KUKA KRL program: Milling_8_4.src

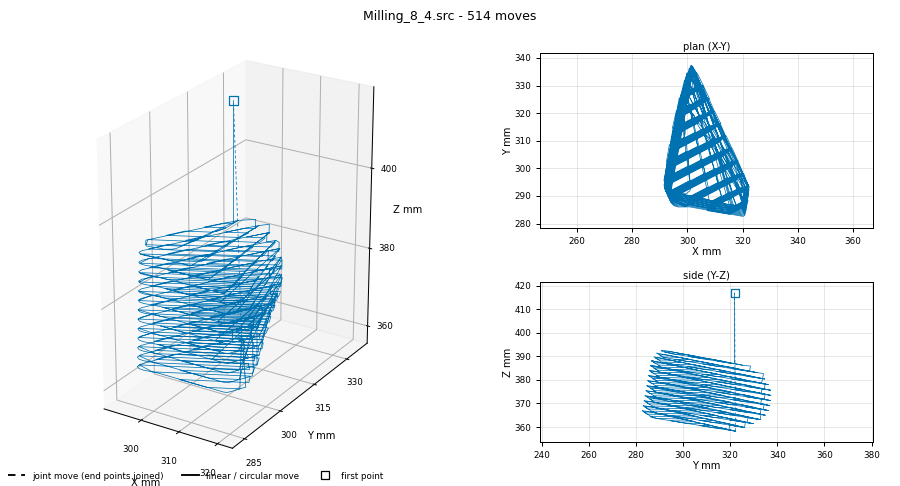
[picture p0: tool path of Milling_8_4.src, 514 of 516 moves have a stored position in this frame; points joined in program order, loops and branches not executed]
&ACCESS RVP
&REL 1
&PARAM TEMPLATE = C:\KRC\Roboter\Template\vorgabe
&PARAM EDITMASK = *
DEF Milling_8_4 ( )


;FOLD INI
;FOLD BASISTECH INI
GLOBAL INTERRUPT DECL 3 WHEN $STOPMESS==TRUE DO IR_STOPM ( )
INTERRUPT ON 3
BAS (#INITMOV,0 )
;ENDFOLD (BASISTECH INI)
;ENDFOLD (INI)

;FOLD STARTPOSITION - BASE IS 0, TOOL IS 5, SPEED IS 15%, POSITION IS A1 5,A2 -90,A3 100,A4 5,A5 -10,A6 -5,E1 0,E2 0,E3 0,E4 0
$BWDSTART = FALSE
PDAT_ACT = {VEL 15,ACC 100,APO_DIST 50}
FDAT_ACT = {TOOL_NO 5,BASE_NO 0,IPO_FRAME #BASE}
BAS (#PTP_PARAMS,15)
PTP  {A1 5,A2 -90,A3 100,A4 5,A5 -10,A6 -5,E1 0,E2 0,E3 0,E4 0}
;ENDFOLD

;FOLD LIN SPEED IS 0.1 m/sec, INTERPOLATION SETTINGS IN FOLD
$VEL.CP=0.1
$ADVANCE=3
;ENDFOLD

BAS(#VEL_PTP,2)
PTP {X 297.852, Y 321.837, Z 416.933, A -65.265, B 78.944, C -140.572, E1 0, E2 0, E3 0, E4 0, S 'B010'}
$VEL.CP=0.012
LIN {X 297.852, Y 321.837, Z 386.933, A -65.265, B 78.944, C -140.572, E1 0, E2 0, E3 0, E4 0}
LIN {X 295.987, Y 320.861, Z 386.954, A -65.265, B 78.944, C -140.572, E1 0, E2 0, E3 0, E4 0}
LIN {X 294.555, Y 314.544, Z 387.958, A -65.265, B 78.944, C -140.572, E1 0, E2 0, E3 0, E4 0}
LIN {X 298.939, Y 316.84, Z 387.909, A -65.265, B 78.944, C -140.572, E1 0, E2 0, E3 0, E4 0}
LIN {X 298.897, Y 311.252, Z 388.897, A -65.265, B 78.944, C -140.572, E1 0, E2 0, E3 0, E4 0}
LIN {X 293.416, Y 308.381, Z 388.959, A -65.265, B 78.944, C -140.572, E1 0, E2 0, E3 0, E4 0}
LIN {X 292.389, Y 302.277, Z 389.958, A -65.265, B 78.944, C -140.572, E1 0, E2 0, E3 0, E4 0}
LIN {X 299.803, Y 306.16, Z 389.875, A -65.265, B 78.944, C -140.572, E1 0, E2 0, E3 0, E4 0}
LIN {X 300.521, Y 300.97, Z 390.855, A -65.265, B 78.944, C -140.572, E1 0, E2 0, E3 0, E4 0}
LIN {X 291.565, Y 296.279, Z 390.955, A -65.265, B 78.944, C -140.572, E1 0, E2 0, E3 0, E4 0}
LIN {X 293.945, Y 291.959, Z 391.916, A -65.265, B 78.944, C -140.572, E1 0, E2 0, E3 0, E4 0}
LIN {X 300.779, Y 295.539, Z 391.84, A -65.265, B 78.944, C -140.572, E1 0, E2 0, E3 0, E4 0}
LIN {X 296.996, Y 325.233, Z 386.261, A -65.265, B 78.944, C -140.572, E1 0, E2 0, E3 0, E4 0}
LIN {X 291.482, Y 295.499, Z 391.087, A -65.265, B 78.944, C -140.572, E1 0, E2 0, E3 0, E4 0}
LIN {X 294.103, Y 291.625, Z 391.989, A -65.265, B 78.944, C -140.572, E1 0, E2 0, E3 0, E4 0}
LIN {X 294.812, Y 290.922, Z 392.171, A -65.265, B 78.944, C -140.572, E1 0, E2 0, E3 0, E4 0}
LIN {X 298.459, Y 290.964, Z 392.462, A -65.265, B 78.944, C -140.572, E1 0, E2 0, E3 0, E4 0}
LIN {X 299.412, Y 290.71, Z 392.585, A -65.265, B 78.944, C -140.572, E1 0, E2 0, E3 0, E4 0}
LIN {X 300.839, Y 291.808, Z 392.507, A -65.265, B 78.944, C -140.572, E1 0, E2 0, E3 0, E4 0}
LIN {X 301.22, Y 292.929, Z 392.339, A -65.265, B 78.944, C -140.572, E1 0, E2 0, E3 0, E4 0}
LIN {X 299.581, Y 309.004, Z 389.352, A -65.265, B 78.944, C -140.572, E1 0, E2 0, E3 0, E4 0}
LIN {X 298.847, Y 311.367, Z 388.873, A -65.265, B 78.944, C -140.572, E1 0, E2 0, E3 0, E4 0}
LIN {X 299.224, Y 312.814, Z 388.647, A -65.265, B 78.944, C -140.572, E1 0, E2 0, E3 0, E4 0}
LIN {X 298.944, Y 316.962, Z 387.888, A -65.265, B 78.944, C -140.572, E1 0, E2 0, E3 0, E4 0}
LIN {X 296.996, Y 325.233, Z 386.261, A -65.265, B 78.944, C -140.572, E1 0, E2 0, E3 0, E4 0}
LIN {X 299.671, Y 328.593, Z 385.883, A -65.265, B 78.944, C -140.572, E1 0, E2 0, E3 0, E4 0}
LIN {X 299.845, Y 328.214, Z 383.749, A -65.265, B 78.944, C -140.572, E1 0, E2 0, E3 0, E4 0}
LIN {X 297.836, Y 327.162, Z 383.772, A -65.265, B 78.944, C -140.572, E1 0, E2 0, E3 0, E4 0}
LIN {X 296.213, Y 320.745, Z 384.778, A -65.265, B 78.944, C -140.572, E1 0, E2 0, E3 0, E4 0}
LIN {X 301.047, Y 323.278, Z 384.724, A -65.265, B 78.944, C -140.572, E1 0, E2 0, E3 0, E4 0}
LIN {X 301.749, Y 318.079, Z 385.704, A -65.265, B 78.944, C -140.572, E1 0, E2 0, E3 0, E4 0}
LIN {X 294.77, Y 314.424, Z 385.782, A -65.265, B 78.944, C -140.572, E1 0, E2 0, E3 0, E4 0}
LIN {X 293.654, Y 308.273, Z 386.783, A -65.265, B 78.944, C -140.572, E1 0, E2 0, E3 0, E4 0}
LIN {X 302.541, Y 312.927, Z 386.683, A -65.265, B 78.944, C -140.572, E1 0, E2 0, E3 0, E4 0}
LIN {X 303.726, Y 307.981, Z 387.658, A -65.265, B 78.944, C -140.572, E1 0, E2 0, E3 0, E4 0}
LIN {X 292.608, Y 302.158, Z 387.782, A -65.265, B 78.944, C -140.572, E1 0, E2 0, E3 0, E4 0}
LIN {X 291.745, Y 296.14, Z 388.78, A -65.265, B 78.944, C -140.572, E1 0, E2 0, E3 0, E4 0}
LIN {X 305.193, Y 303.183, Z 388.629, A -65.265, B 78.944, C -140.572, E1 0, E2 0, E3 0, E4 0}
LIN {X 306.408, Y 298.253, Z 389.603, A -65.265, B 78.944, C -140.572, E1 0, E2 0, E3 0, E4 0}
LIN {X 292.898, Y 291.177, Z 389.755, A -65.265, B 78.944, C -140.572, E1 0, E2 0, E3 0, E4 0}
LIN {X 301.236, Y 289.978, Z 390.649, A -65.265, B 78.944, C -140.572, E1 0, E2 0, E3 0, E4 0}
LIN {X 307.526, Y 293.272, Z 390.579, A -65.265, B 78.944, C -140.572, E1 0, E2 0, E3 0, E4 0}
LIN {X 298.826, Y 331.411, Z 383.099, A -65.265, B 78.944, C -140.572, E1 0, E2 0, E3 0, E4 0}
LIN {X 297.438, Y 325.863, Z 383.97, A -65.265, B 78.944, C -140.572, E1 0, E2 0, E3 0, E4 0}
LIN {X 291.516, Y 293.899, Z 389.159, A -65.265, B 78.944, C -140.572, E1 0, E2 0, E3 0, E4 0}
LIN {X 291.916, Y 292.132, Z 389.505, A -65.265, B 78.944, C -140.572, E1 0, E2 0, E3 0, E4 0}
LIN {X 293.141, Y 290.966, Z 389.812, A -65.265, B 78.944, C -140.572, E1 0, E2 0, E3 0, E4 0}
LIN {X 294.578, Y 290.537, Z 390.005, A -65.265, B 78.944, C -140.572, E1 0, E2 0, E3 0, E4 0}
LIN {X 298.633, Y 290.585, Z 390.328, A -65.265, B 78.944, C -140.572, E1 0, E2 0, E3 0, E4 0}
LIN {X 306.184, Y 288.971, Z 391.232, A -65.265, B 78.944, C -140.572, E1 0, E2 0, E3 0, E4 0}
LIN {X 307.849, Y 288.642, Z 391.427, A -65.265, B 78.944, C -140.572, E1 0, E2 0, E3 0, E4 0}
LIN {X 303.748, Y 307.894, Z 387.675, A -65.265, B 78.944, C -140.572, E1 0, E2 0, E3 0, E4 0}
LIN {X 303.252, Y 309.872, Z 387.283, A -65.265, B 78.944, C -140.572, E1 0, E2 0, E3 0, E4 0}
LIN {X 303.261, Y 309.968, Z 387.267, A -65.265, B 78.944, C -140.572, E1 0, E2 0, E3 0, E4 0}
LIN {X 298.826, Y 331.411, Z 383.099, A -65.265, B 78.944, C -140.572, E1 0, E2 0, E3 0, E4 0}
LIN {X 300.023, Y 334.111, Z 382.718, A -65.265, B 78.944, C -140.572, E1 0, E2 0, E3 0, E4 0}
LIN {X 300.198, Y 333.732, Z 380.584, A -65.265, B 78.944, C -140.572, E1 0, E2 0, E3 0, E4 0}
LIN {X 299.57, Y 333.403, Z 380.591, A -65.265, B 78.944, C -140.572, E1 0, E2 0, E3 0, E4 0}
LIN {X 298.085, Y 327.059, Z 381.596, A -65.265, B 78.944, C -140.572, E1 0, E2 0, E3 0, E4 0}
LIN {X 301.963, Y 329.09, Z 381.552, A -65.265, B 78.944, C -140.572, E1 0, E2 0, E3 0, E4 0}
LIN {X 303.417, Y 324.285, Z 382.524, A -65.265, B 78.944, C -140.572, E1 0, E2 0, E3 0, E4 0}
LIN {X 296.435, Y 320.628, Z 382.602, A -65.265, B 78.944, C -140.572, E1 0, E2 0, E3 0, E4 0}
LIN {X 294.986, Y 314.303, Z 383.606, A -65.265, B 78.944, C -140.572, E1 0, E2 0, E3 0, E4 0}
LIN {X 304.624, Y 319.351, Z 383.498, A -65.265, B 78.944, C -140.572, E1 0, E2 0, E3 0, E4 0}
LIN {X 305.837, Y 314.42, Z 384.473, A -65.265, B 78.944, C -140.572, E1 0, E2 0, E3 0, E4 0}
LIN {X 293.892, Y 308.164, Z 384.606, A -65.265, B 78.944, C -140.572, E1 0, E2 0, E3 0, E4 0}
LIN {X 292.827, Y 302.039, Z 385.606, A -65.265, B 78.944, C -140.572, E1 0, E2 0, E3 0, E4 0}
LIN {X 307.214, Y 309.575, Z 385.445, A -65.265, B 78.944, C -140.572, E1 0, E2 0, E3 0, E4 0}
LIN {X 308.472, Y 304.667, Z 386.419, A -65.265, B 78.944, C -140.572, E1 0, E2 0, E3 0, E4 0}
LIN {X 291.926, Y 296.001, Z 386.604, A -65.265, B 78.944, C -140.572, E1 0, E2 0, E3 0, E4 0}
LIN {X 292.915, Y 290.953, Z 387.581, A -65.265, B 78.944, C -140.572, E1 0, E2 0, E3 0, E4 0}
LIN {X 310.061, Y 299.933, Z 387.389, A -65.265, B 78.944, C -140.572, E1 0, E2 0, E3 0, E4 0}
LIN {X 311.293, Y 295.012, Z 388.363, A -65.265, B 78.944, C -140.572, E1 0, E2 0, E3 0, E4 0}
LIN {X 301.09, Y 289.668, Z 388.477, A -65.265, B 78.944, C -140.572, E1 0, E2 0, E3 0, E4 0}
LIN {X 308.786, Y 288.132, Z 389.379, A -65.265, B 78.944, C -140.572, E1 0, E2 0, E3 0, E4 0}
LIN {X 312.319, Y 289.983, Z 389.339, A -65.265, B 78.944, C -140.572, E1 0, E2 0, E3 0, E4 0}
LIN {X 299.903, Y 334.57, Z 380.411, A -65.265, B 78.944, C -140.572, E1 0, E2 0, E3 0, E4 0}
LIN {X 297.613, Y 325.485, Z 381.836, A -65.265, B 78.944, C -140.572, E1 0, E2 0, E3 0, E4 0}
LIN {X 291.69, Y 293.52, Z 387.025, A -65.265, B 78.944, C -140.572, E1 0, E2 0, E3 0, E4 0}
LIN {X 292.09, Y 291.753, Z 387.371, A -65.265, B 78.944, C -140.572, E1 0, E2 0, E3 0, E4 0}
LIN {X 293.316, Y 290.587, Z 387.678, A -65.265, B 78.944, C -140.572, E1 0, E2 0, E3 0, E4 0}
LIN {X 294.753, Y 290.159, Z 387.872, A -65.265, B 78.944, C -140.572, E1 0, E2 0, E3 0, E4 0}
LIN {X 298.808, Y 290.207, Z 388.195, A -65.265, B 78.944, C -140.572, E1 0, E2 0, E3 0, E4 0}
LIN {X 312.65, Y 287.569, Z 389.795, A -65.265, B 78.944, C -140.572, E1 0, E2 0, E3 0, E4 0}
LIN {X 312.907, Y 287.55, Z 389.819, A -65.265, B 78.944, C -140.572, E1 0, E2 0, E3 0, E4 0}
LIN {X 306.404, Y 312.498, Z 384.86, A -65.265, B 78.944, C -140.572, E1 0, E2 0, E3 0, E4 0}
LIN {X 304.977, Y 316.033, Z 384.116, A -65.265, B 78.944, C -140.572, E1 0, E2 0, E3 0, E4 0}
LIN {X 299.903, Y 334.57, Z 380.411, A -65.265, B 78.944, C -140.572, E1 0, E2 0, E3 0, E4 0}
LIN {X 299.65, Y 333.681, Z 380.548, A -65.265, B 78.944, C -140.572, E1 0, E2 0, E3 0, E4 0}
LIN {X 299.824, Y 333.303, Z 378.415, A -65.265, B 78.944, C -140.572, E1 0, E2 0, E3 0, E4 0}
LIN {X 301.62, Y 334.244, Z 378.395, A -65.265, B 78.944, C -140.572, E1 0, E2 0, E3 0, E4 0}
LIN {X 303.356, Y 329.586, Z 379.363, A -65.265, B 78.944, C -140.572, E1 0, E2 0, E3 0, E4 0}
LIN {X 298.333, Y 326.956, Z 379.419, A -65.265, B 78.944, C -140.572, E1 0, E2 0, E3 0, E4 0}
LIN {X 296.657, Y 320.511, Z 380.426, A -65.265, B 78.944, C -140.572, E1 0, E2 0, E3 0, E4 0}
LIN {X 304.962, Y 324.861, Z 380.333, A -65.265, B 78.944, C -140.572, E1 0, E2 0, E3 0, E4 0}
LIN {X 306.594, Y 320.15, Z 381.303, A -65.265, B 78.944, C -140.572, E1 0, E2 0, E3 0, E4 0}
LIN {X 295.237, Y 314.201, Z 381.43, A -65.265, B 78.944, C -140.572, E1 0, E2 0, E3 0, E4 0}
LIN {X 294.131, Y 308.055, Z 382.43, A -65.265, B 78.944, C -140.572, E1 0, E2 0, E3 0, E4 0}
LIN {X 308.144, Y 315.395, Z 382.273, A -65.265, B 78.944, C -140.572, E1 0, E2 0, E3 0, E4 0}
LIN {X 309.483, Y 310.529, Z 383.246, A -65.265, B 78.944, C -140.572, E1 0, E2 0, E3 0, E4 0}
LIN {X 293.046, Y 301.921, Z 383.43, A -65.265, B 78.944, C -140.572, E1 0, E2 0, E3 0, E4 0}
LIN {X 292.106, Y 295.862, Z 384.428, A -65.265, B 78.944, C -140.572, E1 0, E2 0, E3 0, E4 0}
LIN {X 310.958, Y 305.736, Z 384.217, A -65.265, B 78.944, C -140.572, E1 0, E2 0, E3 0, E4 0}
LIN {X 312.946, Y 301.21, Z 385.183, A -65.265, B 78.944, C -140.572, E1 0, E2 0, E3 0, E4 0}
LIN {X 292.931, Y 290.728, Z 385.407, A -65.265, B 78.944, C -140.572, E1 0, E2 0, E3 0, E4 0}
LIN {X 300.943, Y 289.358, Z 386.305, A -65.265, B 78.944, C -140.572, E1 0, E2 0, E3 0, E4 0}
LIN {X 314.712, Y 296.569, Z 386.151, A -65.265, B 78.944, C -140.572, E1 0, E2 0, E3 0, E4 0}
LIN {X 316.164, Y 291.763, Z 387.123, A -65.265, B 78.944, C -140.572, E1 0, E2 0, E3 0, E4 0}
LIN {X 308.609, Y 287.806, Z 387.207, A -65.265, B 78.944, C -140.572, E1 0, E2 0, E3 0, E4 0}
LIN {X 316.904, Y 286.584, Z 388.102, A -65.265, B 78.944, C -140.572, E1 0, E2 0, E3 0, E4 0}
LIN {X 317.579, Y 286.938, Z 388.095, A -65.265, B 78.944, C -140.572, E1 0, E2 0, E3 0, E4 0}
LIN {X 300.629, Y 336.129, Z 377.979, A -65.265, B 78.944, C -140.572, E1 0, E2 0, E3 0, E4 0}
LIN {X 297.787, Y 325.106, Z 379.703, A -65.265, B 78.944, C -140.572, E1 0, E2 0, E3 0, E4 0}
LIN {X 291.865, Y 293.141, Z 384.891, A -65.265, B 78.944, C -140.572, E1 0, E2 0, E3 0, E4 0}
LIN {X 292.265, Y 291.374, Z 385.238, A -65.265, B 78.944, C -140.572, E1 0, E2 0, E3 0, E4 0}
LIN {X 293.49, Y 290.209, Z 385.545, A -65.265, B 78.944, C -140.572, E1 0, E2 0, E3 0, E4 0}
LIN {X 294.927, Y 289.78, Z 385.738, A -65.265, B 78.944, C -140.572, E1 0, E2 0, E3 0, E4 0}
LIN {X 298.982, Y 289.828, Z 386.061, A -65.265, B 78.944, C -140.572, E1 0, E2 0, E3 0, E4 0}
LIN {X 317.303, Y 286.491, Z 388.151, A -65.265, B 78.944, C -140.572, E1 0, E2 0, E3 0, E4 0}
LIN {X 317.75, Y 286.429, Z 388.199, A -65.265, B 78.944, C -140.572, E1 0, E2 0, E3 0, E4 0}
LIN {X 316.564, Y 289.217, Z 387.607, A -65.265, B 78.944, C -140.572, E1 0, E2 0, E3 0, E4 0}
LIN {X 316.61, Y 290.09, Z 387.456, A -65.265, B 78.944, C -140.572, E1 0, E2 0, E3 0, E4 0}
LIN {X 312.976, Y 301.173, Z 385.192, A -65.265, B 78.944, C -140.572, E1 0, E2 0, E3 0, E4 0}
LIN {X 312.271, Y 302.03, Z 384.982, A -65.265, B 78.944, C -140.572, E1 0, E2 0, E3 0, E4 0}
LIN {X 300.629, Y 336.129, Z 377.979, A -65.265, B 78.944, C -140.572, E1 0, E2 0, E3 0, E4 0}
LIN {X 302.315, Y 334.844, Z 378.345, A -65.265, B 78.944, C -140.572, E1 0, E2 0, E3 0, E4 0}
LIN {X 302.49, Y 334.466, Z 376.211, A -65.265, B 78.944, C -140.572, E1 0, E2 0, E3 0, E4 0}
LIN {X 300.078, Y 333.202, Z 376.238, A -65.265, B 78.944, C -140.572, E1 0, E2 0, E3 0, E4 0}
LIN {X 298.581, Y 326.852, Z 377.243, A -65.265, B 78.944, C -140.572, E1 0, E2 0, E3 0, E4 0}
LIN {X 304.357, Y 329.877, Z 377.178, A -65.265, B 78.944, C -140.572, E1 0, E2 0, E3 0, E4 0}
LIN {X 306.195, Y 325.274, Z 378.146, A -65.265, B 78.944, C -140.572, E1 0, E2 0, E3 0, E4 0}
LIN {X 296.909, Y 320.41, Z 378.25, A -65.265, B 78.944, C -140.572, E1 0, E2 0, E3 0, E4 0}
LIN {X 295.477, Y 314.094, Z 379.253, A -65.265, B 78.944, C -140.572, E1 0, E2 0, E3 0, E4 0}
LIN {X 307.903, Y 320.601, Z 379.114, A -65.265, B 78.944, C -140.572, E1 0, E2 0, E3 0, E4 0}
LIN {X 309.612, Y 315.93, Z 380.083, A -65.265, B 78.944, C -140.572, E1 0, E2 0, E3 0, E4 0}
LIN {X 294.362, Y 307.943, Z 380.254, A -65.265, B 78.944, C -140.572, E1 0, E2 0, E3 0, E4 0}
LIN {X 293.273, Y 301.806, Z 381.254, A -65.265, B 78.944, C -140.572, E1 0, E2 0, E3 0, E4 0}
LIN {X 311.168, Y 311.178, Z 381.054, A -65.265, B 78.944, C -140.572, E1 0, E2 0, E3 0, E4 0}
LIN {X 312.979, Y 306.561, Z 382.021, A -65.265, B 78.944, C -140.572, E1 0, E2 0, E3 0, E4 0}
LIN {X 292.287, Y 295.723, Z 382.253, A -65.265, B 78.944, C -140.572, E1 0, E2 0, E3 0, E4 0}
LIN {X 292.947, Y 290.503, Z 383.233, A -65.265, B 78.944, C -140.572, E1 0, E2 0, E3 0, E4 0}
LIN {X 315.04, Y 302.074, Z 382.986, A -65.265, B 78.944, C -140.572, E1 0, E2 0, E3 0, E4 0}
LIN {X 317.063, Y 297.567, Z 383.951, A -65.265, B 78.944, C -140.572, E1 0, E2 0, E3 0, E4 0}
LIN {X 300.798, Y 289.048, Z 384.133, A -65.265, B 78.944, C -140.572, E1 0, E2 0, E3 0, E4 0}
LIN {X 308.452, Y 287.49, Z 385.036, A -65.265, B 78.944, C -140.572, E1 0, E2 0, E3 0, E4 0}
LIN {X 318.657, Y 292.835, Z 384.921, A -65.265, B 78.944, C -140.572, E1 0, E2 0, E3 0, E4 0}
LIN {X 319.625, Y 287.776, Z 385.898, A -65.265, B 78.944, C -140.572, E1 0, E2 0, E3 0, E4 0}
LIN {X 316.766, Y 286.278, Z 385.93, A -65.265, B 78.944, C -140.572, E1 0, E2 0, E3 0, E4 0}
LIN {X 301.169, Y 337.121, Z 375.632, A -65.265, B 78.944, C -140.572, E1 0, E2 0, E3 0, E4 0}
LIN {X 297.962, Y 324.728, Z 377.569, A -65.265, B 78.944, C -140.572, E1 0, E2 0, E3 0, E4 0}
LIN {X 292.039, Y 292.762, Z 382.758, A -65.265, B 78.944, C -140.572, E1 0, E2 0, E3 0, E4 0}
LIN {X 292.439, Y 290.995, Z 383.104, A -65.265, B 78.944, C -140.572, E1 0, E2 0, E3 0, E4 0}
LIN {X 293.665, Y 289.83, Z 383.411, A -65.265, B 78.944, C -140.572, E1 0, E2 0, E3 0, E4 0}
LIN {X 295.101, Y 289.402, Z 383.605, A -65.265, B 78.944, C -140.572, E1 0, E2 0, E3 0, E4 0}
LIN {X 299.156, Y 289.45, Z 383.928, A -65.265, B 78.944, C -140.572, E1 0, E2 0, E3 0, E4 0}
LIN {X 318.437, Y 286.008, Z 386.115, A -65.265, B 78.944, C -140.572, E1 0, E2 0, E3 0, E4 0}
LIN {X 319.132, Y 286.229, Z 386.132, A -65.265, B 78.944, C -140.572, E1 0, E2 0, E3 0, E4 0}
LIN {X 319.161, Y 286.27, Z 386.128, A -65.265, B 78.944, C -140.572, E1 0, E2 0, E3 0, E4 0}
LIN {X 319.732, Y 288.464, Z 385.785, A -65.265, B 78.944, C -140.572, E1 0, E2 0, E3 0, E4 0}
LIN {X 319.691, Y 288.513, Z 385.773, A -65.265, B 78.944, C -140.572, E1 0, E2 0, E3 0, E4 0}
LIN {X 319.887, Y 289.583, Z 385.599, A -65.265, B 78.944, C -140.572, E1 0, E2 0, E3 0, E4 0}
LIN {X 317.767, Y 296.066, Z 384.275, A -65.265, B 78.944, C -140.572, E1 0, E2 0, E3 0, E4 0}
LIN {X 315.303, Y 301.274, Z 383.149, A -65.265, B 78.944, C -140.572, E1 0, E2 0, E3 0, E4 0}
LIN {X 301.338, Y 336.638, Z 375.732, A -65.265, B 78.944, C -140.572, E1 0, E2 0, E3 0, E4 0}
LIN {X 301.339, Y 336.701, Z 375.72, A -65.265, B 78.944, C -140.572, E1 0, E2 0, E3 0, E4 0}
LIN {X 301.169, Y 337.121, Z 375.632, A -65.265, B 78.944, C -140.572, E1 0, E2 0, E3 0, E4 0}
LIN {X 300.157, Y 333.48, Z 376.195, A -65.265, B 78.944, C -140.572, E1 0, E2 0, E3 0, E4 0}
LIN {X 300.331, Y 333.102, Z 374.062, A -65.265, B 78.944, C -140.572, E1 0, E2 0, E3 0, E4 0}
LIN {X 303.138, Y 334.572, Z 374.03, A -65.265, B 78.944, C -140.572, E1 0, E2 0, E3 0, E4 0}
LIN {X 305.038, Y 330, Z 374.997, A -65.265, B 78.944, C -140.572, E1 0, E2 0, E3 0, E4 0}
LIN {X 298.825, Y 326.746, Z 375.066, A -65.265, B 78.944, C -140.572, E1 0, E2 0, E3 0, E4 0}
LIN {X 297.192, Y 320.324, Z 376.073, A -65.265, B 78.944, C -140.572, E1 0, E2 0, E3 0, E4 0}
LIN {X 306.857, Y 325.386, Z 375.965, A -65.265, B 78.944, C -140.572, E1 0, E2 0, E3 0, E4 0}
LIN {X 308.596, Y 320.731, Z 376.933, A -65.265, B 78.944, C -140.572, E1 0, E2 0, E3 0, E4 0}
LIN {X 295.718, Y 313.986, Z 377.077, A -65.265, B 78.944, C -140.572, E1 0, E2 0, E3 0, E4 0}
LIN {X 294.583, Y 307.825, Z 378.078, A -65.265, B 78.944, C -140.572, E1 0, E2 0, E3 0, E4 0}
LIN {X 310.607, Y 316.218, Z 377.898, A -65.265, B 78.944, C -140.572, E1 0, E2 0, E3 0, E4 0}
LIN {X 312.442, Y 311.612, Z 378.866, A -65.265, B 78.944, C -140.572, E1 0, E2 0, E3 0, E4 0}
LIN {X 293.506, Y 301.695, Z 379.078, A -65.265, B 78.944, C -140.572, E1 0, E2 0, E3 0, E4 0}
LIN {X 292.468, Y 295.584, Z 380.077, A -65.265, B 78.944, C -140.572, E1 0, E2 0, E3 0, E4 0}
LIN {X 314.348, Y 307.044, Z 379.832, A -65.265, B 78.944, C -140.572, E1 0, E2 0, E3 0, E4 0}
LIN {X 316.395, Y 302.55, Z 380.797, A -65.265, B 78.944, C -140.572, E1 0, E2 0, E3 0, E4 0}
LIN {X 292.963, Y 290.278, Z 381.059, A -65.265, B 78.944, C -140.572, E1 0, E2 0, E3 0, E4 0}
LIN {X 300.652, Y 288.738, Z 381.961, A -65.265, B 78.944, C -140.572, E1 0, E2 0, E3 0, E4 0}
LIN {X 318.267, Y 297.964, Z 381.764, A -65.265, B 78.944, C -140.572, E1 0, E2 0, E3 0, E4 0}
LIN {X 319.989, Y 293.299, Z 382.733, A -65.265, B 78.944, C -140.572, E1 0, E2 0, E3 0, E4 0}
LIN {X 308.298, Y 287.176, Z 382.864, A -65.265, B 78.944, C -140.572, E1 0, E2 0, E3 0, E4 0}
LIN {X 316.628, Y 285.972, Z 383.758, A -65.265, B 78.944, C -140.572, E1 0, E2 0, E3 0, E4 0}
LIN {X 319.84, Y 287.655, Z 383.722, A -65.265, B 78.944, C -140.572, E1 0, E2 0, E3 0, E4 0}
LIN {X 301.46, Y 337.237, Z 373.42, A -65.265, B 78.944, C -140.572, E1 0, E2 0, E3 0, E4 0}
LIN {X 298.136, Y 324.349, Z 375.436, A -65.265, B 78.944, C -140.572, E1 0, E2 0, E3 0, E4 0}
LIN {X 292.213, Y 292.384, Z 380.624, A -65.265, B 78.944, C -140.572, E1 0, E2 0, E3 0, E4 0}
LIN {X 292.614, Y 290.617, Z 380.971, A -65.265, B 78.944, C -140.572, E1 0, E2 0, E3 0, E4 0}
LIN {X 293.839, Y 289.451, Z 381.278, A -65.265, B 78.944, C -140.572, E1 0, E2 0, E3 0, E4 0}
LIN {X 295.276, Y 289.023, Z 381.471, A -65.265, B 78.944, C -140.572, E1 0, E2 0, E3 0, E4 0}
LIN {X 299.331, Y 289.071, Z 381.794, A -65.265, B 78.944, C -140.572, E1 0, E2 0, E3 0, E4 0}
LIN {X 318.611, Y 285.629, Z 383.981, A -65.265, B 78.944, C -140.572, E1 0, E2 0, E3 0, E4 0}
LIN {X 319.306, Y 285.85, Z 383.999, A -65.265, B 78.944, C -140.572, E1 0, E2 0, E3 0, E4 0}
LIN {X 319.336, Y 285.891, Z 383.994, A -65.265, B 78.944, C -140.572, E1 0, E2 0, E3 0, E4 0}
LIN {X 319.907, Y 288.086, Z 383.651, A -65.265, B 78.944, C -140.572, E1 0, E2 0, E3 0, E4 0}
LIN {X 319.866, Y 288.134, Z 383.639, A -65.265, B 78.944, C -140.572, E1 0, E2 0, E3 0, E4 0}
LIN {X 320.382, Y 290.88, Z 383.194, A -65.265, B 78.944, C -140.572, E1 0, E2 0, E3 0, E4 0}
LIN {X 320.685, Y 291.937, Z 383.031, A -65.265, B 78.944, C -140.572, E1 0, E2 0, E3 0, E4 0}
LIN {X 308.836, Y 320.346, Z 377.021, A -65.265, B 78.944, C -140.572, E1 0, E2 0, E3 0, E4 0}
LIN {X 308.633, Y 320.593, Z 376.96, A -65.265, B 78.944, C -140.572, E1 0, E2 0, E3 0, E4 0}
LIN {X 301.46, Y 337.237, Z 373.42, A -65.265, B 78.944, C -140.572, E1 0, E2 0, E3 0, E4 0}
LIN {X 303.163, Y 334.821, Z 373.988, A -65.265, B 78.944, C -140.572, E1 0, E2 0, E3 0, E4 0}
LIN {X 303.338, Y 334.443, Z 371.855, A -65.265, B 78.944, C -140.572, E1 0, E2 0, E3 0, E4 0}
LIN {X 300.585, Y 333.001, Z 371.885, A -65.265, B 78.944, C -140.572, E1 0, E2 0, E3 0, E4 0}
LIN {X 299.064, Y 326.638, Z 372.89, A -65.265, B 78.944, C -140.572, E1 0, E2 0, E3 0, E4 0}
LIN {X 305.518, Y 330.018, Z 372.818, A -65.265, B 78.944, C -140.572, E1 0, E2 0, E3 0, E4 0}
LIN {X 307.258, Y 325.363, Z 373.786, A -65.265, B 78.944, C -140.572, E1 0, E2 0, E3 0, E4 0}
LIN {X 297.428, Y 320.215, Z 373.896, A -65.265, B 78.944, C -140.572, E1 0, E2 0, E3 0, E4 0}
LIN {X 295.958, Y 313.878, Z 374.901, A -65.265, B 78.944, C -140.572, E1 0, E2 0, E3 0, E4 0}
LIN {X 309.234, Y 320.832, Z 374.752, A -65.265, B 78.944, C -140.572, E1 0, E2 0, E3 0, E4 0}
LIN {X 311.279, Y 316.336, Z 375.717, A -65.265, B 78.944, C -140.572, E1 0, E2 0, E3 0, E4 0}
LIN {X 294.803, Y 307.707, Z 375.902, A -65.265, B 78.944, C -140.572, E1 0, E2 0, E3 0, E4 0}
LIN {X 293.74, Y 301.583, Z 376.901, A -65.265, B 78.944, C -140.572, E1 0, E2 0, E3 0, E4 0}
LIN {X 313.122, Y 311.735, Z 376.684, A -65.265, B 78.944, C -140.572, E1 0, E2 0, E3 0, E4 0}
LIN {X 315.239, Y 307.278, Z 377.649, A -65.265, B 78.944, C -140.572, E1 0, E2 0, E3 0, E4 0}
LIN {X 292.648, Y 295.446, Z 377.901, A -65.265, B 78.944, C -140.572, E1 0, E2 0, E3 0, E4 0}
LIN {X 292.979, Y 290.052, Z 378.886, A -65.265, B 78.944, C -140.572, E1 0, E2 0, E3 0, E4 0}
LIN {X 317.273, Y 302.776, Z 378.614, A -65.265, B 78.944, C -140.572, E1 0, E2 0, E3 0, E4 0}
LIN {X 319.125, Y 298.18, Z 379.581, A -65.265, B 78.944, C -140.572, E1 0, E2 0, E3 0, E4 0}
LIN {X 300.505, Y 288.428, Z 379.789, A -65.265, B 78.944, C -140.572, E1 0, E2 0, E3 0, E4 0}
LIN {X 308.145, Y 286.862, Z 380.692, A -65.265, B 78.944, C -140.572, E1 0, E2 0, E3 0, E4 0}
LIN {X 320.921, Y 293.554, Z 380.549, A -65.265, B 78.944, C -140.572, E1 0, E2 0, E3 0, E4 0}
LIN {X 320.054, Y 287.534, Z 381.546, A -65.265, B 78.944, C -140.572, E1 0, E2 0, E3 0, E4 0}
LIN {X 316.49, Y 285.667, Z 381.586, A -65.265, B 78.944, C -140.572, E1 0, E2 0, E3 0, E4 0}
LIN {X 301.674, Y 337.061, Z 371.254, A -65.265, B 78.944, C -140.572, E1 0, E2 0, E3 0, E4 0}
LIN {X 298.31, Y 323.97, Z 373.302, A -65.265, B 78.944, C -140.572, E1 0, E2 0, E3 0, E4 0}
LIN {X 292.388, Y 292.005, Z 378.491, A -65.265, B 78.944, C -140.572, E1 0, E2 0, E3 0, E4 0}
LIN {X 292.788, Y 290.238, Z 378.837, A -65.265, B 78.944, C -140.572, E1 0, E2 0, E3 0, E4 0}
LIN {X 294.014, Y 289.073, Z 379.144, A -65.265, B 78.944, C -140.572, E1 0, E2 0, E3 0, E4 0}
LIN {X 295.45, Y 288.644, Z 379.338, A -65.265, B 78.944, C -140.572, E1 0, E2 0, E3 0, E4 0}
LIN {X 299.505, Y 288.692, Z 379.661, A -65.265, B 78.944, C -140.572, E1 0, E2 0, E3 0, E4 0}
LIN {X 318.786, Y 285.251, Z 381.848, A -65.265, B 78.944, C -140.572, E1 0, E2 0, E3 0, E4 0}
LIN {X 319.481, Y 285.471, Z 381.865, A -65.265, B 78.944, C -140.572, E1 0, E2 0, E3 0, E4 0}
LIN {X 319.51, Y 285.513, Z 381.86, A -65.265, B 78.944, C -140.572, E1 0, E2 0, E3 0, E4 0}
LIN {X 320.081, Y 287.707, Z 381.518, A -65.265, B 78.944, C -140.572, E1 0, E2 0, E3 0, E4 0}
LIN {X 320.04, Y 287.755, Z 381.506, A -65.265, B 78.944, C -140.572, E1 0, E2 0, E3 0, E4 0}
LIN {X 320.557, Y 290.501, Z 381.061, A -65.265, B 78.944, C -140.572, E1 0, E2 0, E3 0, E4 0}
LIN {X 321.169, Y 292.964, Z 380.674, A -65.265, B 78.944, C -140.572, E1 0, E2 0, E3 0, E4 0}
LIN {X 301.674, Y 337.061, Z 371.254, A -65.265, B 78.944, C -140.572, E1 0, E2 0, E3 0, E4 0}
LIN {X 300.664, Y 333.279, Z 371.843, A -65.265, B 78.944, C -140.572, E1 0, E2 0, E3 0, E4 0}
LIN {X 300.839, Y 332.9, Z 369.709, A -65.265, B 78.944, C -140.572, E1 0, E2 0, E3 0, E4 0}
LIN {X 303.587, Y 334.34, Z 369.678, A -65.265, B 78.944, C -140.572, E1 0, E2 0, E3 0, E4 0}
LIN {X 305.802, Y 329.933, Z 370.641, A -65.265, B 78.944, C -140.572, E1 0, E2 0, E3 0, E4 0}
LIN {X 299.304, Y 326.53, Z 370.714, A -65.265, B 78.944, C -140.572, E1 0, E2 0, E3 0, E4 0}
LIN {X 297.652, Y 320.099, Z 371.72, A -65.265, B 78.944, C -140.572, E1 0, E2 0, E3 0, E4 0}
LIN {X 307.697, Y 325.36, Z 371.608, A -65.265, B 78.944, C -140.572, E1 0, E2 0, E3 0, E4 0}
LIN {X 309.695, Y 320.839, Z 372.573, A -65.265, B 78.944, C -140.572, E1 0, E2 0, E3 0, E4 0}
LIN {X 296.199, Y 313.771, Z 372.725, A -65.265, B 78.944, C -140.572, E1 0, E2 0, E3 0, E4 0}
LIN {X 295.024, Y 307.589, Z 373.726, A -65.265, B 78.944, C -140.572, E1 0, E2 0, E3 0, E4 0}
LIN {X 311.836, Y 316.395, Z 373.537, A -65.265, B 78.944, C -140.572, E1 0, E2 0, E3 0, E4 0}
LIN {X 313.74, Y 311.825, Z 374.504, A -65.265, B 78.944, C -140.572, E1 0, E2 0, E3 0, E4 0}
LIN {X 293.973, Y 301.472, Z 374.725, A -65.265, B 78.944, C -140.572, E1 0, E2 0, E3 0, E4 0}
LIN {X 292.832, Y 295.308, Z 375.726, A -65.265, B 78.944, C -140.572, E1 0, E2 0, E3 0, E4 0}
LIN {X 315.726, Y 307.299, Z 375.47, A -65.265, B 78.944, C -140.572, E1 0, E2 0, E3 0, E4 0}
LIN {X 317.862, Y 302.851, Z 376.434, A -65.265, B 78.944, C -140.572, E1 0, E2 0, E3 0, E4 0}
LIN {X 292.996, Y 289.828, Z 376.712, A -65.265, B 78.944, C -140.572, E1 0, E2 0, E3 0, E4 0}
LIN {X 300.369, Y 288.123, Z 377.617, A -65.265, B 78.944, C -140.572, E1 0, E2 0, E3 0, E4 0}
LIN {X 319.757, Y 298.277, Z 377.4, A -65.265, B 78.944, C -140.572, E1 0, E2 0, E3 0, E4 0}
LIN {X 321.581, Y 293.666, Z 378.368, A -65.265, B 78.944, C -140.572, E1 0, E2 0, E3 0, E4 0}
LIN {X 307.991, Y 286.549, Z 378.52, A -65.265, B 78.944, C -140.572, E1 0, E2 0, E3 0, E4 0}
LIN {X 316.351, Y 285.361, Z 379.414, A -65.265, B 78.944, C -140.572, E1 0, E2 0, E3 0, E4 0}
LIN {X 320.217, Y 287.385, Z 379.371, A -65.265, B 78.944, C -140.572, E1 0, E2 0, E3 0, E4 0}
LIN {X 301.878, Y 336.832, Z 369.096, A -65.265, B 78.944, C -140.572, E1 0, E2 0, E3 0, E4 0}
LIN {X 298.485, Y 323.591, Z 371.169, A -65.265, B 78.944, C -140.572, E1 0, E2 0, E3 0, E4 0}
LIN {X 292.562, Y 291.627, Z 376.357, A -65.265, B 78.944, C -140.572, E1 0, E2 0, E3 0, E4 0}
LIN {X 292.963, Y 289.86, Z 376.704, A -65.265, B 78.944, C -140.572, E1 0, E2 0, E3 0, E4 0}
LIN {X 294.188, Y 288.694, Z 377.01, A -65.265, B 78.944, C -140.572, E1 0, E2 0, E3 0, E4 0}
LIN {X 295.625, Y 288.266, Z 377.204, A -65.265, B 78.944, C -140.572, E1 0, E2 0, E3 0, E4 0}
LIN {X 299.68, Y 288.314, Z 377.527, A -65.265, B 78.944, C -140.572, E1 0, E2 0, E3 0, E4 0}
LIN {X 318.96, Y 284.872, Z 379.714, A -65.265, B 78.944, C -140.572, E1 0, E2 0, E3 0, E4 0}
LIN {X 319.655, Y 285.093, Z 379.732, A -65.265, B 78.944, C -140.572, E1 0, E2 0, E3 0, E4 0}
LIN {X 319.684, Y 285.134, Z 379.727, A -65.265, B 78.944, C -140.572, E1 0, E2 0, E3 0, E4 0}
LIN {X 320.256, Y 287.329, Z 379.384, A -65.265, B 78.944, C -140.572, E1 0, E2 0, E3 0, E4 0}
LIN {X 320.215, Y 287.377, Z 379.372, A -65.265, B 78.944, C -140.572, E1 0, E2 0, E3 0, E4 0}
LIN {X 321.593, Y 293.717, Z 378.36, A -65.265, B 78.944, C -140.572, E1 0, E2 0, E3 0, E4 0}
LIN {X 321.64, Y 293.944, Z 378.323, A -65.265, B 78.944, C -140.572, E1 0, E2 0, E3 0, E4 0}
LIN {X 301.878, Y 336.832, Z 369.096, A -65.265, B 78.944, C -140.572, E1 0, E2 0, E3 0, E4 0}
LIN {X 303.24, Y 334.394, Z 369.64, A -65.265, B 78.944, C -140.572, E1 0, E2 0, E3 0, E4 0}
LIN {X 303.414, Y 334.016, Z 367.507, A -65.265, B 78.944, C -140.572, E1 0, E2 0, E3 0, E4 0}
LIN {X 301.092, Y 332.8, Z 367.533, A -65.265, B 78.944, C -140.572, E1 0, E2 0, E3 0, E4 0}
LIN {X 299.543, Y 326.422, Z 368.538, A -65.265, B 78.944, C -140.572, E1 0, E2 0, E3 0, E4 0}
LIN {X 305.85, Y 329.725, Z 368.467, A -65.265, B 78.944, C -140.572, E1 0, E2 0, E3 0, E4 0}
LIN {X 307.954, Y 325.261, Z 369.432, A -65.265, B 78.944, C -140.572, E1 0, E2 0, E3 0, E4 0}
LIN {X 297.877, Y 319.983, Z 369.544, A -65.265, B 78.944, C -140.572, E1 0, E2 0, E3 0, E4 0}
LIN {X 296.439, Y 313.663, Z 370.548, A -65.265, B 78.944, C -140.572, E1 0, E2 0, E3 0, E4 0}
LIN {X 309.839, Y 320.681, Z 370.398, A -65.265, B 78.944, C -140.572, E1 0, E2 0, E3 0, E4 0}
LIN {X 312.041, Y 316.268, Z 371.362, A -65.265, B 78.944, C -140.572, E1 0, E2 0, E3 0, E4 0}
LIN {X 295.244, Y 307.471, Z 371.55, A -65.265, B 78.944, C -140.572, E1 0, E2 0, E3 0, E4 0}
LIN {X 294.206, Y 301.361, Z 372.549, A -65.265, B 78.944, C -140.572, E1 0, E2 0, E3 0, E4 0}
LIN {X 314.048, Y 311.753, Z 372.327, A -65.265, B 78.944, C -140.572, E1 0, E2 0, E3 0, E4 0}
LIN {X 316.11, Y 307.266, Z 373.292, A -65.265, B 78.944, C -140.572, E1 0, E2 0, E3 0, E4 0}
LIN {X 293.027, Y 295.177, Z 373.55, A -65.265, B 78.944, C -140.572, E1 0, E2 0, E3 0, E4 0}
LIN {X 293.067, Y 289.631, Z 374.538, A -65.265, B 78.944, C -140.572, E1 0, E2 0, E3 0, E4 0}
LIN {X 318.235, Y 302.813, Z 374.256, A -65.265, B 78.944, C -140.572, E1 0, E2 0, E3 0, E4 0}
LIN {X 320.145, Y 298.247, Z 375.222, A -65.265, B 78.944, C -140.572, E1 0, E2 0, E3 0, E4 0}
LIN {X 300.248, Y 287.826, Z 375.445, A -65.265, B 78.944, C -140.572, E1 0, E2 0, E3 0, E4 0}
LIN {X 307.838, Y 286.235, Z 376.348, A -65.265, B 78.944, C -140.572, E1 0, E2 0, E3 0, E4 0}
LIN {X 321.811, Y 293.553, Z 376.192, A -65.265, B 78.944, C -140.572, E1 0, E2 0, E3 0, E4 0}
LIN {X 320.455, Y 287.276, Z 377.195, A -65.265, B 78.944, C -140.572, E1 0, E2 0, E3 0, E4 0}
LIN {X 316.238, Y 285.068, Z 377.242, A -65.265, B 78.944, C -140.572, E1 0, E2 0, E3 0, E4 0}
LIN {X 302.007, Y 336.221, Z 367, A -65.265, B 78.944, C -140.572, E1 0, E2 0, E3 0, E4 0}
LIN {X 298.659, Y 323.213, Z 369.035, A -65.265, B 78.944, C -140.572, E1 0, E2 0, E3 0, E4 0}
LIN {X 292.737, Y 291.248, Z 374.224, A -65.265, B 78.944, C -140.572, E1 0, E2 0, E3 0, E4 0}
LIN {X 293.137, Y 289.481, Z 374.57, A -65.265, B 78.944, C -140.572, E1 0, E2 0, E3 0, E4 0}
LIN {X 294.362, Y 288.315, Z 374.877, A -65.265, B 78.944, C -140.572, E1 0, E2 0, E3 0, E4 0}
LIN {X 295.799, Y 287.887, Z 375.071, A -65.265, B 78.944, C -140.572, E1 0, E2 0, E3 0, E4 0}
LIN {X 299.854, Y 287.935, Z 375.394, A -65.265, B 78.944, C -140.572, E1 0, E2 0, E3 0, E4 0}
LIN {X 319.135, Y 284.494, Z 377.581, A -65.265, B 78.944, C -140.572, E1 0, E2 0, E3 0, E4 0}
LIN {X 319.83, Y 284.714, Z 377.598, A -65.265, B 78.944, C -140.572, E1 0, E2 0, E3 0, E4 0}
LIN {X 319.859, Y 284.755, Z 377.593, A -65.265, B 78.944, C -140.572, E1 0, E2 0, E3 0, E4 0}
LIN {X 320.43, Y 286.95, Z 377.25, A -65.265, B 78.944, C -140.572, E1 0, E2 0, E3 0, E4 0}
LIN {X 320.389, Y 286.998, Z 377.239, A -65.265, B 78.944, C -140.572, E1 0, E2 0, E3 0, E4 0}
LIN {X 321.799, Y 293.51, Z 376.198, A -65.265, B 78.944, C -140.572, E1 0, E2 0, E3 0, E4 0}
LIN {X 321.946, Y 294.035, Z 376.117, A -65.265, B 78.944, C -140.572, E1 0, E2 0, E3 0, E4 0}
LIN {X 302.007, Y 336.221, Z 367, A -65.265, B 78.944, C -140.572, E1 0, E2 0, E3 0, E4 0}
LIN {X 301.172, Y 333.078, Z 367.49, A -65.265, B 78.944, C -140.572, E1 0, E2 0, E3 0, E4 0}
LIN {X 301.346, Y 332.699, Z 365.356, A -65.265, B 78.944, C -140.572, E1 0, E2 0, E3 0, E4 0}
LIN {X 302.848, Y 333.486, Z 365.339, A -65.265, B 78.944, C -140.572, E1 0, E2 0, E3 0, E4 0}
LIN {X 305.209, Y 329.156, Z 366.301, A -65.265, B 78.944, C -140.572, E1 0, E2 0, E3 0, E4 0}
LIN {X 299.782, Y 326.314, Z 366.362, A -65.265, B 78.944, C -140.572, E1 0, E2 0, E3 0, E4 0}
LIN {X 298.102, Y 319.867, Z 367.368, A -65.265, B 78.944, C -140.572, E1 0, E2 0, E3 0, E4 0}
LIN {X 307.384, Y 324.729, Z 367.264, A -65.265, B 78.944, C -140.572, E1 0, E2 0, E3 0, E4 0}
LIN {X 309.517, Y 320.28, Z 368.228, A -65.265, B 78.944, C -140.572, E1 0, E2 0, E3 0, E4 0}
LIN {X 296.646, Y 313.538, Z 368.372, A -65.265, B 78.944, C -140.572, E1 0, E2 0, E3 0, E4 0}
LIN {X 295.465, Y 307.353, Z 369.373, A -65.265, B 78.944, C -140.572, E1 0, E2 0, E3 0, E4 0}
LIN {X 311.643, Y 315.827, Z 369.192, A -65.265, B 78.944, C -140.572, E1 0, E2 0, E3 0, E4 0}
LIN {X 313.873, Y 311.428, Z 370.155, A -65.265, B 78.944, C -140.572, E1 0, E2 0, E3 0, E4 0}
LIN {X 294.439, Y 301.249, Z 370.373, A -65.265, B 78.944, C -140.572, E1 0, E2 0, E3 0, E4 0}
LIN {X 293.245, Y 295.057, Z 371.374, A -65.265, B 78.944, C -140.572, E1 0, E2 0, E3 0, E4 0}
LIN {X 316.272, Y 307.118, Z 371.116, A -65.265, B 78.944, C -140.572, E1 0, E2 0, E3 0, E4 0}
LIN {X 318.304, Y 302.616, Z 372.081, A -65.265, B 78.944, C -140.572, E1 0, E2 0, E3 0, E4 0}
LIN {X 293.197, Y 289.466, Z 372.362, A -65.265, B 78.944, C -140.572, E1 0, E2 0, E3 0, E4 0}
LIN {X 300.127, Y 287.529, Z 373.273, A -65.265, B 78.944, C -140.572, E1 0, E2 0, E3 0, E4 0}
LIN {X 320.371, Y 298.132, Z 373.046, A -65.265, B 78.944, C -140.572, E1 0, E2 0, E3 0, E4 0}
LIN {X 322.063, Y 293.452, Z 374.015, A -65.265, B 78.944, C -140.572, E1 0, E2 0, E3 0, E4 0}
LIN {X 307.684, Y 285.921, Z 374.176, A -65.265, B 78.944, C -140.572, E1 0, E2 0, E3 0, E4 0}
LIN {X 316.083, Y 284.753, Z 375.07, A -65.265, B 78.944, C -140.572, E1 0, E2 0, E3 0, E4 0}
LIN {X 320.693, Y 287.168, Z 375.018, A -65.265, B 78.944, C -140.572, E1 0, E2 0, E3 0, E4 0}
LIN {X 301.952, Y 334.849, Z 365.024, A -65.265, B 78.944, C -140.572, E1 0, E2 0, E3 0, E4 0}
LIN {X 298.834, Y 322.834, Z 366.901, A -65.265, B 78.944, C -140.572, E1 0, E2 0, E3 0, E4 0}
LIN {X 292.911, Y 290.869, Z 372.09, A -65.265, B 78.944, C -140.572, E1 0, E2 0, E3 0, E4 0}
LIN {X 293.311, Y 289.102, Z 372.436, A -65.265, B 78.944, C -140.572, E1 0, E2 0, E3 0, E4 0}
LIN {X 294.537, Y 287.937, Z 372.743, A -65.265, B 78.944, C -140.572, E1 0, E2 0, E3 0, E4 0}
LIN {X 295.974, Y 287.508, Z 372.937, A -65.265, B 78.944, C -140.572, E1 0, E2 0, E3 0, E4 0}
LIN {X 300.029, Y 287.557, Z 373.26, A -65.265, B 78.944, C -140.572, E1 0, E2 0, E3 0, E4 0}
LIN {X 319.309, Y 284.115, Z 375.447, A -65.265, B 78.944, C -140.572, E1 0, E2 0, E3 0, E4 0}
LIN {X 320.004, Y 284.335, Z 375.465, A -65.265, B 78.944, C -140.572, E1 0, E2 0, E3 0, E4 0}
LIN {X 320.033, Y 284.377, Z 375.46, A -65.265, B 78.944, C -140.572, E1 0, E2 0, E3 0, E4 0}
LIN {X 320.605, Y 286.571, Z 375.117, A -65.265, B 78.944, C -140.572, E1 0, E2 0, E3 0, E4 0}
LIN {X 320.564, Y 286.619, Z 375.105, A -65.265, B 78.944, C -140.572, E1 0, E2 0, E3 0, E4 0}
LIN {X 321.941, Y 292.96, Z 374.093, A -65.265, B 78.944, C -140.572, E1 0, E2 0, E3 0, E4 0}
LIN {X 322.147, Y 293.754, Z 373.969, A -65.265, B 78.944, C -140.572, E1 0, E2 0, E3 0, E4 0}
LIN {X 301.952, Y 334.849, Z 365.024, A -65.265, B 78.944, C -140.572, E1 0, E2 0, E3 0, E4 0}
LIN {X 301.57, Y 333.053, Z 365.312, A -65.265, B 78.944, C -140.572, E1 0, E2 0, E3 0, E4 0}
LIN {X 301.744, Y 332.674, Z 363.178, A -65.265, B 78.944, C -140.572, E1 0, E2 0, E3 0, E4 0}
LIN {X 301.6, Y 332.598, Z 363.18, A -65.265, B 78.944, C -140.572, E1 0, E2 0, E3 0, E4 0}
LIN {X 300.022, Y 326.206, Z 364.185, A -65.265, B 78.944, C -140.572, E1 0, E2 0, E3 0, E4 0}
LIN {X 303.925, Y 328.25, Z 364.141, A -65.265, B 78.944, C -140.572, E1 0, E2 0, E3 0, E4 0}
LIN {X 305.94, Y 323.739, Z 365.107, A -65.265, B 78.944, C -140.572, E1 0, E2 0, E3 0, E4 0}
LIN {X 298.327, Y 319.751, Z 365.192, A -65.265, B 78.944, C -140.572, E1 0, E2 0, E3 0, E4 0}
LIN {X 296.846, Y 313.409, Z 366.197, A -65.265, B 78.944, C -140.572, E1 0, E2 0, E3 0, E4 0}
LIN {X 308.313, Y 319.415, Z 366.068, A -65.265, B 78.944, C -140.572, E1 0, E2 0, E3 0, E4 0}
LIN {X 310.654, Y 315.075, Z 367.03, A -65.265, B 78.944, C -140.572, E1 0, E2 0, E3 0, E4 0}
LIN {X 295.685, Y 307.235, Z 367.198, A -65.265, B 78.944, C -140.572, E1 0, E2 0, E3 0, E4 0}
LIN {X 294.672, Y 301.138, Z 368.197, A -65.265, B 78.944, C -140.572, E1 0, E2 0, E3 0, E4 0}
LIN {X 313.104, Y 310.792, Z 367.99, A -65.265, B 78.944, C -140.572, E1 0, E2 0, E3 0, E4 0}
LIN {X 315.475, Y 306.467, Z 368.952, A -65.265, B 78.944, C -140.572, E1 0, E2 0, E3 0, E4 0}
LIN {X 293.477, Y 294.945, Z 369.198, A -65.265, B 78.944, C -140.572, E1 0, E2 0, E3 0, E4 0}
LIN {X 293.327, Y 289.301, Z 370.188, A -65.265, B 78.944, C -140.572, E1 0, E2 0, E3 0, E4 0}
LIN {X 317.942, Y 302.193, Z 369.912, A -65.265, B 78.944, C -140.572, E1 0, E2 0, E3 0, E4 0}
LIN {X 320.263, Y 297.842, Z 370.874, A -65.265, B 78.944, C -140.572, E1 0, E2 0, E3 0, E4 0}
LIN {X 299.793, Y 287.12, Z 371.103, A -65.265, B 78.944, C -140.572, E1 0, E2 0, E3 0, E4 0}
LIN {X 307.521, Y 285.602, Z 372.004, A -65.265, B 78.944, C -140.572, E1 0, E2 0, E3 0, E4 0}
LIN {X 322.306, Y 293.346, Z 371.839, A -65.265, B 78.944, C -140.572, E1 0, E2 0, E3 0, E4 0}
LIN {X 320.901, Y 287.043, Z 372.842, A -65.265, B 78.944, C -140.572, E1 0, E2 0, E3 0, E4 0}
LIN {X 315.862, Y 284.404, Z 372.899, A -65.265, B 78.944, C -140.572, E1 0, E2 0, E3 0, E4 0}
LIN {X 301.658, Y 332.804, Z 363.148, A -65.265, B 78.944, C -140.572, E1 0, E2 0, E3 0, E4 0}
LIN {X 299.008, Y 322.456, Z 364.768, A -65.265, B 78.944, C -140.572, E1 0, E2 0, E3 0, E4 0}
LIN {X 293.086, Y 290.491, Z 369.957, A -65.265, B 78.944, C -140.572, E1 0, E2 0, E3 0, E4 0}
LIN {X 293.486, Y 288.724, Z 370.303, A -65.265, B 78.944, C -140.572, E1 0, E2 0, E3 0, E4 0}
LIN {X 294.711, Y 287.558, Z 370.61, A -65.265, B 78.944, C -140.572, E1 0, E2 0, E3 0, E4 0}
LIN {X 296.148, Y 287.13, Z 370.803, A -65.265, B 78.944, C -140.572, E1 0, E2 0, E3 0, E4 0}
LIN {X 300.203, Y 287.178, Z 371.126, A -65.265, B 78.944, C -140.572, E1 0, E2 0, E3 0, E4 0}
LIN {X 319.484, Y 283.736, Z 373.313, A -65.265, B 78.944, C -140.572, E1 0, E2 0, E3 0, E4 0}
LIN {X 320.178, Y 283.957, Z 373.331, A -65.265, B 78.944, C -140.572, E1 0, E2 0, E3 0, E4 0}
LIN {X 320.208, Y 283.998, Z 373.326, A -65.265, B 78.944, C -140.572, E1 0, E2 0, E3 0, E4 0}
LIN {X 320.779, Y 286.193, Z 372.983, A -65.265, B 78.944, C -140.572, E1 0, E2 0, E3 0, E4 0}
LIN {X 320.738, Y 286.241, Z 372.972, A -65.265, B 78.944, C -140.572, E1 0, E2 0, E3 0, E4 0}
LIN {X 322.116, Y 292.581, Z 371.959, A -65.265, B 78.944, C -140.572, E1 0, E2 0, E3 0, E4 0}
LIN {X 322.311, Y 293.336, Z 371.841, A -65.265, B 78.944, C -140.572, E1 0, E2 0, E3 0, E4 0}
LIN {X 301.658, Y 332.804, Z 363.148, A -65.265, B 78.944, C -140.572, E1 0, E2 0, E3 0, E4 0}
LIN {X 302.151, Y 327.557, Z 364.119, A -65.265, B 78.944, C -140.572, E1 0, E2 0, E3 0, E4 0}
LIN {X 302.325, Y 327.179, Z 361.986, A -65.265, B 78.944, C -140.572, E1 0, E2 0, E3 0, E4 0}
LIN {X 300.261, Y 326.097, Z 362.009, A -65.265, B 78.944, C -140.572, E1 0, E2 0, E3 0, E4 0}
LIN {X 298.551, Y 319.636, Z 363.016, A -65.265, B 78.944, C -140.572, E1 0, E2 0, E3 0, E4 0}
LIN {X 304.361, Y 322.678, Z 362.951, A -65.265, B 78.944, C -140.572, E1 0, E2 0, E3 0, E4 0}
LIN {X 306.663, Y 318.318, Z 363.913, A -65.265, B 78.944, C -140.572, E1 0, E2 0, E3 0, E4 0}
LIN {X 297.046, Y 313.281, Z 364.021, A -65.265, B 78.944, C -140.572, E1 0, E2 0, E3 0, E4 0}
LIN {X 295.906, Y 307.117, Z 365.021, A -65.265, B 78.944, C -140.572, E1 0, E2 0, E3 0, E4 0}
LIN {X 309.488, Y 314.231, Z 364.869, A -65.265, B 78.944, C -140.572, E1 0, E2 0, E3 0, E4 0}
LIN {X 312.258, Y 310.115, Z 365.826, A -65.265, B 78.944, C -140.572, E1 0, E2 0, E3 0, E4 0}
LIN {X 294.905, Y 301.027, Z 366.02, A -65.265, B 78.944, C -140.572, E1 0, E2 0, E3 0, E4 0}
LIN {X 293.709, Y 294.833, Z 367.022, A -65.265, B 78.944, C -140.572, E1 0, E2 0, E3 0, E4 0}
LIN {X 314.519, Y 305.733, Z 366.789, A -65.265, B 78.944, C -140.572, E1 0, E2 0, E3 0, E4 0}
LIN {X 317.186, Y 301.563, Z 367.747, A -65.265, B 78.944, C -140.572, E1 0, E2 0, E3 0, E4 0}
LIN {X 293.457, Y 289.135, Z 368.012, A -65.265, B 78.944, C -140.572, E1 0, E2 0, E3 0, E4 0}
LIN {X 299.593, Y 286.782, Z 368.932, A -65.265, B 78.944, C -140.572, E1 0, E2 0, E3 0, E4 0}
LIN {X 319.834, Y 297.384, Z 368.705, A -65.265, B 78.944, C -140.572, E1 0, E2 0, E3 0, E4 0}
LIN {X 322.039, Y 292.972, Z 369.668, A -65.265, B 78.944, C -140.572, E1 0, E2 0, E3 0, E4 0}
LIN {X 307.354, Y 285.281, Z 369.833, A -65.265, B 78.944, C -140.572, E1 0, E2 0, E3 0, E4 0}
LIN {X 315.642, Y 284.055, Z 370.728, A -65.265, B 78.944, C -140.572, E1 0, E2 0, E3 0, E4 0}
LIN {X 321.106, Y 286.917, Z 370.667, A -65.265, B 78.944, C -140.572, E1 0, E2 0, E3 0, E4 0}
LIN {X 301.081, Y 329.789, Z 361.421, A -65.265, B 78.944, C -140.572, E1 0, E2 0, E3 0, E4 0}
LIN {X 299.183, Y 322.077, Z 362.634, A -65.265, B 78.944, C -140.572, E1 0, E2 0, E3 0, E4 0}
LIN {X 293.26, Y 290.112, Z 367.823, A -65.265, B 78.944, C -140.572, E1 0, E2 0, E3 0, E4 0}
LIN {X 293.66, Y 288.345, Z 368.169, A -65.265, B 78.944, C -140.572, E1 0, E2 0, E3 0, E4 0}
LIN {X 294.886, Y 287.18, Z 368.476, A -65.265, B 78.944, C -140.572, E1 0, E2 0, E3 0, E4 0}
LIN {X 296.322, Y 286.751, Z 368.67, A -65.265, B 78.944, C -140.572, E1 0, E2 0, E3 0, E4 0}
LIN {X 300.378, Y 286.799, Z 368.993, A -65.265, B 78.944, C -140.572, E1 0, E2 0, E3 0, E4 0}
LIN {X 319.658, Y 283.358, Z 371.18, A -65.265, B 78.944, C -140.572, E1 0, E2 0, E3 0, E4 0}
LIN {X 320.353, Y 283.578, Z 371.198, A -65.265, B 78.944, C -140.572, E1 0, E2 0, E3 0, E4 0}
LIN {X 320.382, Y 283.619, Z 371.193, A -65.265, B 78.944, C -140.572, E1 0, E2 0, E3 0, E4 0}
LIN {X 320.953, Y 285.814, Z 370.85, A -65.265, B 78.944, C -140.572, E1 0, E2 0, E3 0, E4 0}
LIN {X 320.912, Y 285.862, Z 370.838, A -65.265, B 78.944, C -140.572, E1 0, E2 0, E3 0, E4 0}
LIN {X 322.29, Y 292.203, Z 369.825, A -65.265, B 78.944, C -140.572, E1 0, E2 0, E3 0, E4 0}
LIN {X 322.331, Y 292.404, Z 369.793, A -65.265, B 78.944, C -140.572, E1 0, E2 0, E3 0, E4 0}
LIN {X 305.684, Y 319.501, Z 363.623, A -65.265, B 78.944, C -140.572, E1 0, E2 0, E3 0, E4 0}
LIN {X 301.081, Y 329.789, Z 361.421, A -65.265, B 78.944, C -140.572, E1 0, E2 0, E3 0, E4 0}
LIN {X 300.452, Y 326.434, Z 361.965, A -65.265, B 78.944, C -140.572, E1 0, E2 0, E3 0, E4 0}
LIN {X 300.626, Y 326.055, Z 359.831, A -65.265, B 78.944, C -140.572, E1 0, E2 0, E3 0, E4 0}
LIN {X 300.492, Y 325.985, Z 359.833, A -65.265, B 78.944, C -140.572, E1 0, E2 0, E3 0, E4 0}
LIN {X 298.78, Y 319.522, Z 360.84, A -65.265, B 78.944, C -140.572, E1 0, E2 0, E3 0, E4 0}
LIN {X 302.912, Y 321.686, Z 360.794, A -65.265, B 78.944, C -140.572, E1 0, E2 0, E3 0, E4 0}
LIN {X 305.382, Y 317.413, Z 361.754, A -65.265, B 78.944, C -140.572, E1 0, E2 0, E3 0, E4 0}
LIN {X 297.246, Y 313.152, Z 361.845, A -65.265, B 78.944, C -140.572, E1 0, E2 0, E3 0, E4 0}
LIN {X 296.129, Y 307, Z 362.845, A -65.265, B 78.944, C -140.572, E1 0, E2 0, E3 0, E4 0}
LIN {X 308.413, Y 313.434, Z 362.708, A -65.265, B 78.944, C -140.572, E1 0, E2 0, E3 0, E4 0}
LIN {X 311.232, Y 309.344, Z 363.664, A -65.265, B 78.944, C -140.572, E1 0, E2 0, E3 0, E4 0}
LIN {X 295.136, Y 300.914, Z 363.844, A -65.265, B 78.944, C -140.572, E1 0, E2 0, E3 0, E4 0}
LIN {X 293.94, Y 294.721, Z 364.846, A -65.265, B 78.944, C -140.572, E1 0, E2 0, E3 0, E4 0}
LIN {X 313.889, Y 305.17, Z 364.622, A -65.265, B 78.944, C -140.572, E1 0, E2 0, E3 0, E4 0}
LIN {X 316.431, Y 300.934, Z 365.582, A -65.265, B 78.944, C -140.572, E1 0, E2 0, E3 0, E4 0}
LIN {X 293.587, Y 288.969, Z 365.837, A -65.265, B 78.944, C -140.572, E1 0, E2 0, E3 0, E4 0}
LIN {X 299.397, Y 286.446, Z 366.76, A -65.265, B 78.944, C -140.572, E1 0, E2 0, E3 0, E4 0}
LIN {X 319.141, Y 296.788, Z 366.539, A -65.265, B 78.944, C -140.572, E1 0, E2 0, E3 0, E4 0}
LIN {X 321.217, Y 292.308, Z 367.504, A -65.265, B 78.944, C -140.572, E1 0, E2 0, E3 0, E4 0}
LIN {X 307.205, Y 284.969, Z 367.661, A -65.265, B 78.944, C -140.572, E1 0, E2 0, E3 0, E4 0}
LIN {X 315.421, Y 283.706, Z 368.557, A -65.265, B 78.944, C -140.572, E1 0, E2 0, E3 0, E4 0}
LIN {X 321.311, Y 286.791, Z 368.491, A -65.265, B 78.944, C -140.572, E1 0, E2 0, E3 0, E4 0}
LIN {X 300.534, Y 326.194, Z 359.799, A -65.265, B 78.944, C -140.572, E1 0, E2 0, E3 0, E4 0}
LIN {X 299.357, Y 321.698, Z 360.501, A -65.265, B 78.944, C -140.572, E1 0, E2 0, E3 0, E4 0}
LIN {X 293.434, Y 289.734, Z 365.689, A -65.265, B 78.944, C -140.572, E1 0, E2 0, E3 0, E4 0}
LIN {X 293.835, Y 287.967, Z 366.036, A -65.265, B 78.944, C -140.572, E1 0, E2 0, E3 0, E4 0}
LIN {X 295.06, Y 286.801, Z 366.343, A -65.265, B 78.944, C -140.572, E1 0, E2 0, E3 0, E4 0}
LIN {X 296.497, Y 286.372, Z 366.536, A -65.265, B 78.944, C -140.572, E1 0, E2 0, E3 0, E4 0}
LIN {X 300.552, Y 286.42, Z 366.859, A -65.265, B 78.944, C -140.572, E1 0, E2 0, E3 0, E4 0}
LIN {X 319.833, Y 282.979, Z 369.046, A -65.265, B 78.944, C -140.572, E1 0, E2 0, E3 0, E4 0}
LIN {X 320.527, Y 283.199, Z 369.064, A -65.265, B 78.944, C -140.572, E1 0, E2 0, E3 0, E4 0}
LIN {X 320.557, Y 283.241, Z 369.059, A -65.265, B 78.944, C -140.572, E1 0, E2 0, E3 0, E4 0}
LIN {X 321.128, Y 285.436, Z 368.716, A -65.265, B 78.944, C -140.572, E1 0, E2 0, E3 0, E4 0}
LIN {X 321.087, Y 285.483, Z 368.704, A -65.265, B 78.944, C -140.572, E1 0, E2 0, E3 0, E4 0}
LIN {X 321.809, Y 288.846, Z 368.167, A -65.265, B 78.944, C -140.572, E1 0, E2 0, E3 0, E4 0}
LIN {X 322.211, Y 290.672, Z 367.876, A -65.265, B 78.944, C -140.572, E1 0, E2 0, E3 0, E4 0}
LIN {X 320.958, Y 292.686, Z 367.416, A -65.265, B 78.944, C -140.572, E1 0, E2 0, E3 0, E4 0}
LIN {X 320.846, Y 293.283, Z 367.3, A -65.265, B 78.944, C -140.572, E1 0, E2 0, E3 0, E4 0}
LIN {X 306.757, Y 315.781, Z 362.156, A -65.265, B 78.944, C -140.572, E1 0, E2 0, E3 0, E4 0}
LIN {X 306.796, Y 315.824, Z 362.151, A -65.265, B 78.944, C -140.572, E1 0, E2 0, E3 0, E4 0}
LIN {X 304.488, Y 318.457, Z 361.495, A -65.265, B 78.944, C -140.572, E1 0, E2 0, E3 0, E4 0}
LIN {X 300.534, Y 326.194, Z 359.799, A -65.265, B 78.944, C -140.572, E1 0, E2 0, E3 0, E4 0}
LIN {X 298.853, Y 319.796, Z 360.797, A -65.265, B 78.944, C -140.572, E1 0, E2 0, E3 0, E4 0}
LIN {X 299.027, Y 319.418, Z 358.663, A -65.265, B 78.944, C -140.572, E1 0, E2 0, E3 0, E4 0}
LIN {X 301.223, Y 320.568, Z 358.639, A -65.265, B 78.944, C -140.572, E1 0, E2 0, E3 0, E4 0}
LIN {X 304.072, Y 316.493, Z 359.595, A -65.265, B 78.944, C -140.572, E1 0, E2 0, E3 0, E4 0}
LIN {X 297.446, Y 313.023, Z 359.669, A -65.265, B 78.944, C -140.572, E1 0, E2 0, E3 0, E4 0}
LIN {X 296.357, Y 306.886, Z 360.669, A -65.265, B 78.944, C -140.572, E1 0, E2 0, E3 0, E4 0}
LIN {X 306.652, Y 312.279, Z 360.554, A -65.265, B 78.944, C -140.572, E1 0, E2 0, E3 0, E4 0}
LIN {X 310.2, Y 308.57, Z 361.502, A -65.265, B 78.944, C -140.572, E1 0, E2 0, E3 0, E4 0}
LIN {X 295.337, Y 300.786, Z 361.668, A -65.265, B 78.944, C -140.572, E1 0, E2 0, E3 0, E4 0}
LIN {X 294.172, Y 294.609, Z 362.669, A -65.265, B 78.944, C -140.572, E1 0, E2 0, E3 0, E4 0}
LIN {X 312.721, Y 304.324, Z 362.462, A -65.265, B 78.944, C -140.572, E1 0, E2 0, E3 0, E4 0}
LIN {X 315.568, Y 300.249, Z 363.418, A -65.265, B 78.944, C -140.572, E1 0, E2 0, E3 0, E4 0}
LIN {X 293.716, Y 288.804, Z 363.662, A -65.265, B 78.944, C -140.572, E1 0, E2 0, E3 0, E4 0}
LIN {X 299.095, Y 286.055, Z 364.59, A -65.265, B 78.944, C -140.572, E1 0, E2 0, E3 0, E4 0}
LIN {X 318.276, Y 296.101, Z 364.375, A -65.265, B 78.944, C -140.572, E1 0, E2 0, E3 0, E4 0}
LIN {X 320.658, Y 291.782, Z 365.337, A -65.265, B 78.944, C -140.572, E1 0, E2 0, E3 0, E4 0}
LIN {X 307.094, Y 284.678, Z 365.488, A -65.265, B 78.944, C -140.572, E1 0, E2 0, E3 0, E4 0}
LIN {X 315.195, Y 283.354, Z 366.386, A -65.265, B 78.944, C -140.572, E1 0, E2 0, E3 0, E4 0}
LIN {X 321.516, Y 286.665, Z 366.315, A -65.265, B 78.944, C -140.572, E1 0, E2 0, E3 0, E4 0}
LIN {X 299.813, Y 322.187, Z 358.236, A -65.265, B 78.944, C -140.572, E1 0, E2 0, E3 0, E4 0}
LIN {X 299.531, Y 321.32, Z 358.367, A -65.265, B 78.944, C -140.572, E1 0, E2 0, E3 0, E4 0}
LIN {X 293.609, Y 289.355, Z 363.556, A -65.265, B 78.944, C -140.572, E1 0, E2 0, E3 0, E4 0}
LIN {X 294.009, Y 287.588, Z 363.902, A -65.265, B 78.944, C -140.572, E1 0, E2 0, E3 0, E4 0}
LIN {X 295.234, Y 286.422, Z 364.209, A -65.265, B 78.944, C -140.572, E1 0, E2 0, E3 0, E4 0}
LIN {X 296.671, Y 285.994, Z 364.403, A -65.265, B 78.944, C -140.572, E1 0, E2 0, E3 0, E4 0}
LIN {X 300.726, Y 286.042, Z 364.726, A -65.265, B 78.944, C -140.572, E1 0, E2 0, E3 0, E4 0}
LIN {X 320.007, Y 282.6, Z 366.913, A -65.265, B 78.944, C -140.572, E1 0, E2 0, E3 0, E4 0}
LIN {X 320.702, Y 282.821, Z 366.93, A -65.265, B 78.944, C -140.572, E1 0, E2 0, E3 0, E4 0}
LIN {X 320.731, Y 282.862, Z 366.926, A -65.265, B 78.944, C -140.572, E1 0, E2 0, E3 0, E4 0}
LIN {X 321.302, Y 285.057, Z 366.583, A -65.265, B 78.944, C -140.572, E1 0, E2 0, E3 0, E4 0}
LIN {X 321.261, Y 285.105, Z 366.571, A -65.265, B 78.944, C -140.572, E1 0, E2 0, E3 0, E4 0}
LIN {X 321.693, Y 287.562, Z 366.17, A -65.265, B 78.944, C -140.572, E1 0, E2 0, E3 0, E4 0}
LIN {X 321.958, Y 288.392, Z 366.044, A -65.265, B 78.944, C -140.572, E1 0, E2 0, E3 0, E4 0}
LIN {X 305.896, Y 313.139, Z 360.339, A -65.265, B 78.944, C -140.572, E1 0, E2 0, E3 0, E4 0}
LIN {X 305.44, Y 314.61, Z 360.041, A -65.265, B 78.944, C -140.572, E1 0, E2 0, E3 0, E4 0}
LIN {X 302.861, Y 317.919, Z 359.243, A -65.265, B 78.944, C -140.572, E1 0, E2 0, E3 0, E4 0}
LIN {X 302.486, Y 319.118, Z 358.999, A -65.265, B 78.944, C -140.572, E1 0, E2 0, E3 0, E4 0}
LIN {X 299.813, Y 322.187, Z 358.236, A -65.265, B 78.944, C -140.572, E1 0, E2 0, E3 0, E4 0}
PTP {X 297.852, Y 321.837, Z 416.933, A -65.265, B 78.944, C -140.572, E1 0, E2 0, E3 0, E4 0, S 'B010'}
PTP {A1 5, A2 -90, A3 100, A4 5, A5 -10, A6 -5, E1 0, E2 0, E3 0, E4 0} C_PTP

END
